FUNCTION F_LogLA2C 
VAR_INPUT
	eLogLevel		: E_LogLevel;
	sLogger			: T_MaxString;
	sMessage		: T_MaxString;
	aArg1			: ANY;
	aArg2			: ANY;
	iContextBuilder	: I_ContextBuilder;
END_VAR
VAR 
	aEmptyArg		: BYTE;
END_VAR

F_LogA(
	eLogLevel,
	sLogger,
	sMessage,
	2,
	aArg1,
	aArg2,
	aEmptyArg,
	aEmptyArg,
	aEmptyArg,
	aEmptyArg,
	aEmptyArg,
	aEmptyArg,
	aEmptyArg,
	aEmptyArg,
	iContextBuilder
);

END_FUNCTION

(* stored: Version 1.1.0.1, ProductVersion 3.1.4024.0
   POU F_LogLA2C: Id {ec2cad51-d003-46f1-9700-837ab05fb474}, SpecialFunc None *)
